Fanuc KAREL source: kt00208.KL

-- PROVISIONAL review KL for V1013-1; original PC SHA256 b081823f850310bd0aa803070e30b93ba9bbb1b2d27d5dc6c7fdf26e2672b71e
-- Incomplete behavior may be omitted. Consult companion uncertainty JSON. Do not deploy.
PROGRAM KT00208
%NOLOCKGROUP
VAR
  I1 : INTEGER
  OUT : INTEGER
-- UNRESOLVED_DECL H2 type=002017
BEGIN
  -- UNRESOLVED_PC offsets 5-16; opcodes 2E,23
  -- UNRESOLVED_PC offsets 21-35; opcodes 2E,22,9D,33,B4
  -- UNRESOLVED_PC offsets 40-62; opcodes 21,22,9D,33,B3,46,23
  -- UNRESOLVED_PC offsets 67-71; opcodes 7F
END KT00208
